SUBAPPLICATION ACTION_CLIENT_CANCEL_GOAL
  (* Standard: 61499-2 *)
  (* Version 1.0, 2023-03-23, Tim Hesse *)
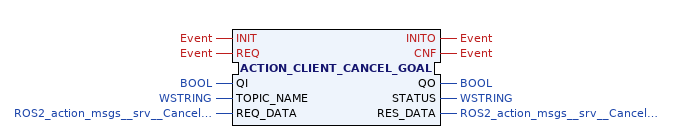
  EVENT_INPUT
    INIT; (* Initialization Request *)
    REQ; (* Normal Execution Request *)
  END_EVENT
  EVENT_OUTPUT
    INITO; (* Initialization Confirm *)
    CNF; (* Execution Confirmation *)
  END_EVENT
  VAR_INPUT
    QI : BOOL; (* Input event qualifier *)
    TOPIC_NAME : WSTRING;
    REQ_DATA : ROS2_action_msgs__srv__CancelGoal__Request;
  END_VAR
  VAR_OUTPUT
    QO : BOOL; (* Output event qualifier *)
    STATUS : WSTRING;
    RES_DATA : ROS2_action_msgs__srv__CancelGoal__Response;
  END_VAR
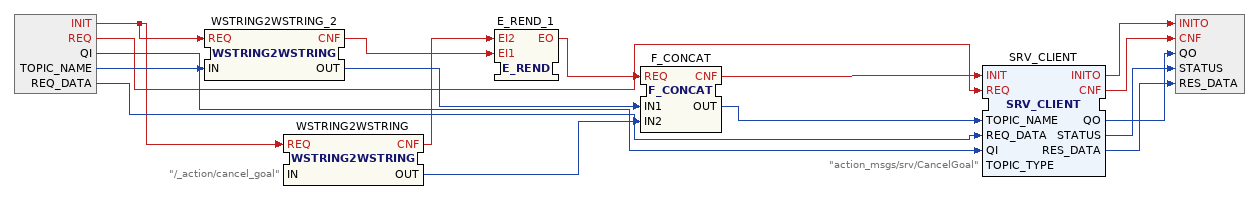
  FBS
    E_REND_1 : E_REND;
    F_CONCAT : F_CONCAT;
    WSTRING2WSTRING_2 : WSTRING2WSTRING;
    WSTRING2WSTRING : WSTRING2WSTRING(IN := "/_action/cancel_goal");
  END_FBS
  SUBAPPS
    SRV_CLIENT : SRV_CLIENT(TOPIC_TYPE := "action_msgs/srv/CancelGoal");
  END_SUBAPPS
  EVENT_CONNECTIONS
    WSTRING2WSTRING.CNF TO E_REND_1.EI2;
    WSTRING2WSTRING_2.CNF TO E_REND_1.EI1;
    E_REND_1.EO TO F_CONCAT.REQ;
    F_CONCAT.CNF TO SRV_CLIENT.INIT;
    INIT TO WSTRING2WSTRING_2.REQ;
    INIT TO WSTRING2WSTRING.REQ;
    REQ TO SRV_CLIENT.REQ;
    SRV_CLIENT.INITO TO INITO;
    SRV_CLIENT.CNF TO CNF;
  END_CONNECTIONS
  DATA_CONNECTIONS
    WSTRING2WSTRING_2.OUT TO F_CONCAT.IN1;
    F_CONCAT.OUT TO SRV_CLIENT.TOPIC_NAME;
    WSTRING2WSTRING.OUT TO F_CONCAT.IN2;
    TOPIC_NAME TO WSTRING2WSTRING_2.IN;
    REQ_DATA TO SRV_CLIENT.REQ_DATA;
    QI TO SRV_CLIENT.QI;
    SRV_CLIENT.QO TO QO;
    SRV_CLIENT.STATUS TO STATUS;
    SRV_CLIENT.RES_DATA TO RES_DATA;
  END_CONNECTIONS
END_SUBAPPLICATION
